FUNCTION_BLOCK TurnOffCommand EXTENDS I_Command
VAR
	_device	:I_Device;
END_VAR

METHOD execute
_device.turnOff();
END_METHOD

METHOD FB_init : BOOL
VAR_INPUT
	bInitRetains : BOOL; // if TRUE, the retain variables are initialized (warm start / cold start)
	bInCopyCode : BOOL;  // if TRUE, the instance afterwards gets moved into the copy code (online change)
	
	device	:I_Device;
END_VAR
THIS^._device := device;
END_METHOD

END_FUNCTION_BLOCK

(* stored: Version 1.1.0.1
   POU TurnOffCommand: Id {7bc8b26d-52a2-4d18-b9a0-dfa25e1824f4}, SpecialFunc None
   Method execute: Id {fb8e3201-89ad-48ff-989e-cad5f6c0930d}
   Method FB_init: Id {a96e9b2b-2a90-446a-8ed0-3f6fb34f6ce1} *)
